(* PLC project motor_1dir_2speed, Dassault Systèmes ControlBuild 2024x *)
(* stored: creationDateTime 2023-10-03T11:13:10-01:00 *)

(* This module simulates the behaviour of a motor with 1 direction and 2 speeds and its electrical control logic. *)
FUNCTION_BLOCK equipment_library.motor_1dir_2speed
  VAR_INPUT
    voltage380 : BOOL := true;
    cmdSupply : BOOL := true;
    sensorSupply : BOOL := true;
  END_VAR
  VAR_INPUT
    highSpeed : BOOL := false;
    lowSpeed : BOOL := false;
  END_VAR
  VAR_OUTPUT
    highSpeedFB : BOOL := false;
    lowSpeedFB : BOOL := false;
    thermal : BOOL := false;
  END_VAR
  VAR_OUTPUT
    speedVal : REAL := 0.0;
    speedPercent : REAL := 0.0;
  END_VAR
  VAR
    increment : REAL := 0.0;
    memoHighSpeed : BOOL := false;
    memoLowSpeed : BOOL := false;
    highSpeedState : BOOL := false;
    lowSpeedState : BOOL := false;
    wantedSpeed : REAL := 0.0;
  END_VAR
  VAR CONSTANT
    nominalTime : REAL := 0.5;
    thermalLogic : BOOL := false;
    highSpeedFBLogic : BOOL := true;
    lowSpeedFBLogic : BOOL := true;
    nominalLowSpeed : REAL := 2500.0;
    nominalHighSpeed : REAL := 5000.0;
  END_VAR
  VAR
    d_locking : BOOL := false;
    v_d_locking : REAL := 0.5;
    d_electrical : BOOL := false;
    v_d_electrical : BOOL := false;
    d_highSpeedFB : BOOL := false;
    v_d_highSpeedFB : BOOL := false;
    d_lowSpeedFB : BOOL := false;
    v_d_lowSpeedFB : BOOL := false;
  END_VAR


ACTION C_source_code:
/* ----------------------------------------------------------------	*/
/* Type : Model of Operative Behaviour					*/
/* Category :  Associations - motors					*/
/* Author : Dassault Systemes						*/
/* Update date : June 2018							*/
/* ----------------------------------------------------------------	*/
/* This module simulates a motor with 1 direction and 2 speeds	*/
/* and its electrical control logic.					*/
/* ----------------------------------------------------------------	*/


/* ----------------------------------------------------------------	*/
/* Management of orders from Control Part					*/
/*	if there is no power supply for command 				*/
/*     the contactors don't understand the control order		*/
/*	The contactors are not mechanically bound.			*/
/* ----------------------------------------------------------------	*/
if (!memoHighSpeed && lowSpeed && cmdSupply) memoLowSpeed = 1;
if (!lowSpeed || !cmdSupply || d_electrical) memoLowSpeed = 0;
if (highSpeed && !memoLowSpeed && cmdSupply) memoHighSpeed = 1;
if (!highSpeed || !cmdSupply || d_electrical) memoHighSpeed = 0;

/* ----------------------------------------------------------------	*/
/* Calculation of the on-state of contactor				*/
/* ----------------------------------------------------------------	*/
highSpeedState=memoHighSpeed & voltage380;
lowSpeedState=memoLowSpeed & voltage380;

/* ----------------------------------------------------------------	*/
/* Management of the speed ramp						*/
/* ----------------------------------------------------------------	*/
if (d_locking)  speedVal = v_d_locking;
else {
	/* Compute the wanted speed according to the state of contactors	*/
	wantedSpeed = 0.0;
	if (highSpeedState) {
		wantedSpeed = nominalHighSpeed;
		if (nominalTime > 0.0)
			increment = (nominalHighSpeed / nominalTime) * (CLOCK_PERIOD/1000000.0);
	}
	else if (lowSpeedState) {
		wantedSpeed = nominalLowSpeed;
		if (nominalTime > 0.0)
			increment = (nominalLowSpeed / nominalTime) * (CLOCK_PERIOD/1000000.0);
	}

	/* Compute speed ramp	*/
	if ( speedVal < wantedSpeed ) {
		speedVal += increment;
		if ( speedVal > wantedSpeed ) speedVal = wantedSpeed;
	}
	if ( speedVal > wantedSpeed ) {
		speedVal -= increment;
		if (speedVal < wantedSpeed) speedVal = wantedSpeed;
	}
}


/* ----------------------------------------------------------------	*/
/* Compute the percentage between the current and nominal speed	*/
/* ----------------------------------------------------------------	*/
if (nominalHighSpeed != 0.0)
	speedPercent = ((speedVal/nominalHighSpeed)*100);

/* ----------------------------------------------------------------	*/
/* Management of the thermal feedback					*/
/* ----------------------------------------------------------------	*/
if (d_electrical) thermal=v_d_electrical;
else
	thermal= ! thermalLogic && sensorSupply;


/* ----------------------------------------------------------------	*/
/* Management of feedback to Control Part					*/
/*     if a fault is required, the contactor feed-back 		*/
/*		 takes a preset state.					*/
/*	if there is no power supply for sensors 				*/
/*         contactor feed-back returns nothing				*/
/*     else contactor feed-back returns the contactor state combined	*/
/*	    with wiring logic.						*/
/* ----------------------------------------------------------------	*/
if (d_highSpeedFB) highSpeedFB = v_d_highSpeedFB;
else 	
	highSpeedFB = (memoHighSpeed ^ ! highSpeedFBLogic) && sensorSupply;


if (d_lowSpeedFB) lowSpeedFB = v_d_lowSpeedFB;
else	
	lowSpeedFB = (memoLowSpeed ^ ! lowSpeedFBLogic) && sensorSupply;
END_ACTION
END_FUNCTION_BLOCK
